// Mitsubishi GX Developer project: 四相八拍步进驱动控制（一）   PLC: FX3U

PROGRAM MAIN
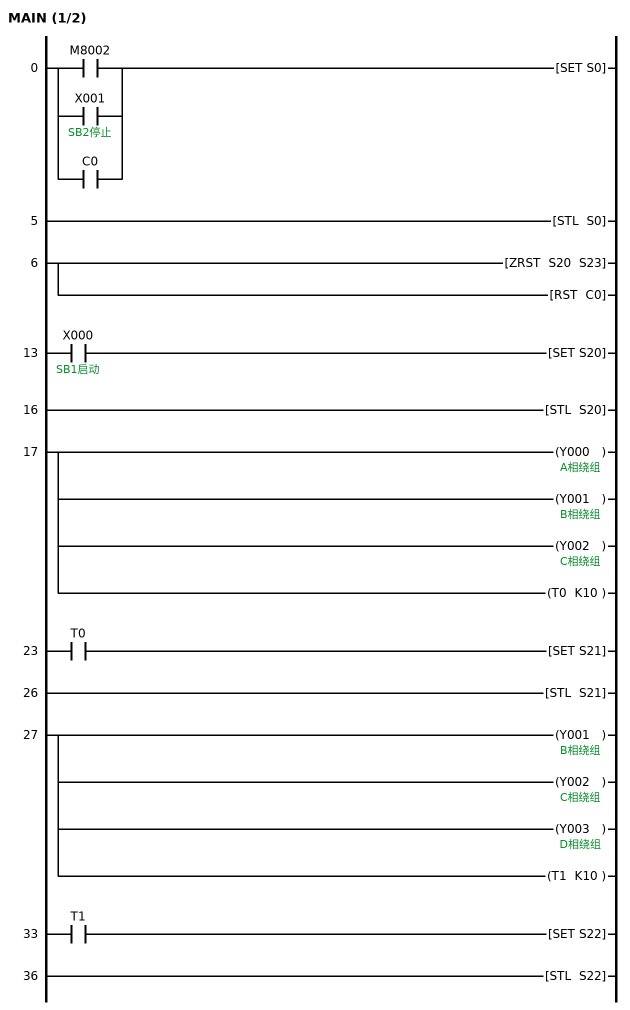
0     LD      M8002
      OR      X001  ; SB2停止
      OR      C0
      SET     S0
5     STL     S0
6     ZRST    S20 S23
      RST     C0
13    LD      X000  ; SB1启动
      SET     S20
16    STL     S20
17    OUT     Y000  ; A相绕组
      OUT     Y001  ; B相绕组
      OUT     Y002  ; C相绕组
      OUT     T0 K10
23    LD      T0
      SET     S21
26    STL     S21
27    OUT     Y001  ; B相绕组
      OUT     Y002  ; C相绕组
      OUT     Y003  ; D相绕组
      OUT     T1 K10
33    LD      T1
      SET     S22
36    STL     S22
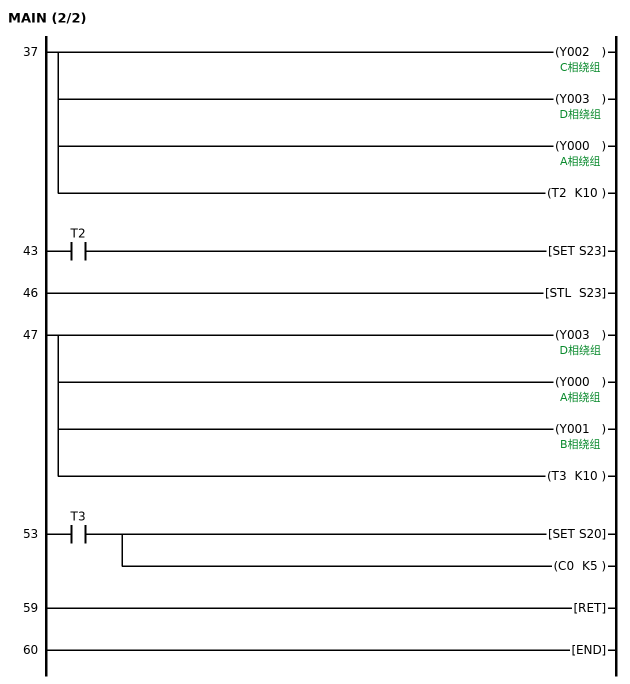
37    OUT     Y002  ; C相绕组
      OUT     Y003  ; D相绕组
      OUT     Y000  ; A相绕组
      OUT     T2 K10
43    LD      T2
      SET     S23
46    STL     S23
47    OUT     Y003  ; D相绕组
      OUT     Y000  ; A相绕组
      OUT     Y001  ; B相绕组
      OUT     T3 K10
53    LD      T3
      SET     S20
      OUT     C0 K5
59    RET
60    END
END_PROGRAM
